KUKA KRL program: WHOLE.src

&ACCESS RV1
&REL 4
&PARAM TEMPLATE = C:\KRC\Roboter\Template\FunctionVorgabe
&PARAM EDITMASK = *
DEFFCT INT WHOLE(VALUE:IN )
  REAL VALUE
  REAL TEMP
  INT RET_VAL

  TEMP = DECIMAL(VALUE)
  RET_VAL = VALUE - TEMP
  RETURN (RET_VAL)
ENDFCT
